FUNCTION_BLOCK NET_VAR_REAL8
VAR_IN_OUT
	X : NET_VAR_DATA;
END_VAR
VAR_INPUT
	IN1 : REAL;
	IN2 : REAL;
	IN3 : REAL;
	IN4 : REAL;
	IN5 : REAL;
	IN6 : REAL;
	IN7 : REAL;
	IN8 : REAL;
END_VAR
VAR_OUTPUT
	OUT1 : REAL;
	OUT2 : REAL;
	OUT3 : REAL;
	OUT4 : REAL;
	OUT5 : REAL;
	OUT6 : REAL;
	OUT7 : REAL;
	OUT8 : REAL;
	ID : BYTE;
END_VAR
VAR
	init : BOOL;
	i : INT;
	i2 : INT;
	index : INT;
	index2 : INT;
	r_dw : DWORD;
	ra : ARRAY[1..8] OF REAL;
END_VAR

(*
version 1.0		15. may. 2011
programmer		ks
tested by			ks

NET_VAR_REAL8 überträgt bidirektional acht REAL-Werte vom Master zum Client
*)

IF NOT init THEN
	init := TRUE;
	X.ID_MAX := X.ID_MAX + USINT#1;
	ID := USINT_TO_BYTE(X.ID_MAX);
END_IF;

IF X.STATE > BYTE#0 AND X.ERROR_ID = BYTE#0 THEN
	index := X.index; (* PCWORX Workaround *)
	IF TO_UINT(index + 34) > X.BUF_SIZE THEN (* ID (1) + TYPE (1) + 8 x REAL (4) *)
		X.ERROR_ID := ID;
	ELSE
		IF X.STATE = BYTE#1 THEN (* Daten schreiben *)
			ra[1] := IN1;
			ra[2] := IN2;
			ra[3] := IN3;
			ra[4] := IN4;
			ra[5] := IN5;
			ra[6] := IN6;
			ra[7] := IN7;
			ra[8] := IN8;
			X.S_BUF.BUFFER[index] := ID; (* ID *)
			index := index + 1;
			X.S_BUF.BUFFER[index] := BYTE#15; (* TYPE REAL8 *)
			index := index + 1;
			FOR i2 := 1 TO 8 DO;
				r_dw := REAL_TO_DW(X:=ra[i2]);
				FOR i := 1 TO 4 DO;
					X.S_BUF.BUFFER[index] := DWORD_TO_BYTE(r_dw);
					r_dw := ROR(r_dw,8);
					index := index + 1;
				END_FOR;
			END_FOR;

		ELSIF X.STATE = BYTE#2 THEN (* Daten lesen *)
			index2 := index + 1; (* PCWORX Workaround *)
			IF X.R_BUF.BUFFER[index] <> ID OR X.R_BUF.BUFFER[index2] <> BYTE#15 THEN (* TYPE REAL8 *)
				X.ERROR_ID := ID;
			ELSE
				index := index + 2;
				FOR i2 := 1 TO 8 DO;
					r_dw := DWORD#0;
					FOR i := 1 TO 4 DO;
						r_dw := r_dw OR BYTE_TO_DWORD(X.R_BUF.BUFFER[index]);
						r_dw := ROR(r_dw,8);
						index := index + 1;
					END_FOR;
					ra[i2] := DW_TO_REAL(X:=r_dw);
				END_FOR;
				OUT1 := ra[1];
				OUT2 := ra[2];
				OUT3 := ra[3];
				OUT4 := ra[4];
				OUT5 := ra[5];
				OUT6 := ra[6];
				OUT7 := ra[7];
				OUT8 := ra[8];
			END_IF;
		END_IF;
		X.index := index;
	END_IF;
END_IF;

(* revision history
ks	15.may. 2011	rev 1.0
	original version

*)

END_FUNCTION_BLOCK

(* stored: Version 1.1.0.1, ProductVersion 3.1.4024.9
   POU NET_VAR_REAL8: Id {c7547c73-5160-45f5-8ac0-1c2118f769d5}, SpecialFunc None *)
